PROGRAM MAIN
VAR
END_VAR

P_Sample();

END_PROGRAM

(* stored: Version 1.1.0.1, ProductVersion 3.1.4024.12
   POU MAIN: Id {8185e429-ba7a-41bc-99f3-636d37d5272b}, SpecialFunc None *)
